SUBAPPLICATION Uebung_011c_AUDI (* Numeric Value Input I3 Durchschleifen auf N3 *)
  (* Standard: 61499-2; Description: Copyright (c) 2023 Meisterschulen am Ostbahnhof This program and the accompanying materials are made available under the terms of the Eclipse Public License 2.0 which is available at https://www.eclipse.org/legal/epl-2.0/ SPDX-License-Identifier: EPL-2.0 *)
  (* Version 1.0, 2026-04-14, Franz Höpfinger, Meisterschulen am Ostbahnhof, initial API and implementation and/or initial documentation *)
  PACKAGE Uebungen;
  IMPORT Uebungen::const::UT::DefaultPool::InputNumber_I3;
  IMPORT Uebungen::const::UT::DefaultPool::OutputNumber_N3;
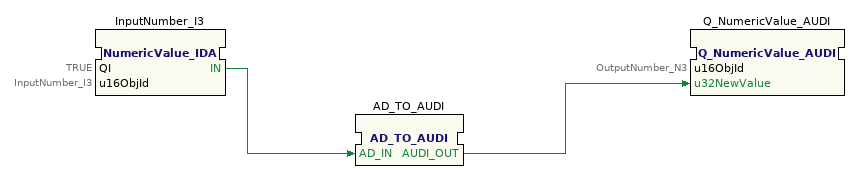
  FBS
    InputNumber_I3 : isobus::UT::io::NumericValue::NumericValue_IDA(QI := TRUE, u16ObjId := InputNumber_I3);
    AD_TO_AUDI : adapter::conversion::unidirectional::AD_TO_AUDI;
    Q_NumericValue_AUDI : isobus::UT::Q::Q_NumericValue_AUDI(u16ObjId := OutputNumber_N3);
  END_FBS
  ADAPTER_CONNECTIONS
    AD_TO_AUDI.AUDI_OUT TO Q_NumericValue_AUDI.u32NewValue;
    InputNumber_I3.IN TO AD_TO_AUDI.AD_IN;
  END_CONNECTIONS
END_SUBAPPLICATION
